FUNCTION_BLOCK F_LEN_ARRAY (* Returns the length of the dimension of the given array *)
  (* Standard: 61499-2; Classification: array function; Description: Copyright (c) 2026 Martin Melik Merkumians, Demmler Andreas Fahrzeugbau This program and the accompanying materials are made available under the terms of the Eclipse Public License 2.0 which is available at https://www.eclipse.org/legal/epl-2.0/ *)
  (* Version 1.1, 2026-04-11, Franz Höpfinger, Demmler Andreas Fahrzeugbau, make same as F_nn_BOUND *)
  (* Version 1.0, 2026-03-25, Martin Melik Merkumians *)
  PACKAGE eclipse4diac::utils::arrays;
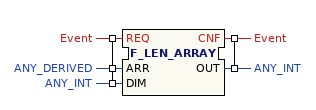
  EVENT_INPUT
    REQ WITH ARR, DIM; (* Service Request *)
  END_EVENT
  EVENT_OUTPUT
    CNF WITH OUT; (* Confirmation of Requested Service *)
  END_EVENT
  VAR_INPUT
    ARR : ANY_DERIVED; (* input array *)
    DIM : ANY_INT := DINT#1; (* Selects array dimension to get the length from, defaults to first dimension *)
  END_VAR
  VAR_OUTPUT
    OUT : ANY_INT; (* Length of the selected array dimension *)
  END_VAR
  EC_STATES
    REQ : REQ -> CNF;
  END_STATES
  ALGORITHM REQ IN ST:
OUT := ADD(SUB(UPPER_BOUND(ARR, DIM), LOWER_BOUND(ARR, DIM)), 1);
  END_ALGORITHM
END_FUNCTION_BLOCK
